SUBAPPLICATION VDS_Auswahl (* Waehlt per Button die satellitengestuetzte Geschwindigkeit (VDS) als Quelle aus, merkt sich die Auswahl persistent im NVS, setzt bei Auswahl die anderen Quellen zurueck und liefert die VDS-Sensordaten nach aussen *)
  (* Standard: 61499-2 *)
  (* Version 1.0, 2026-08-27, Franz *)
  PACKAGE FBs::Baumsetzer::func::Automatik;
  IMPORT NVS_Keys::Key_VDS_Store;
  IMPORT isobus::UT::io::Button::ButtonActivationCode::BT_RELEASED_UNLATCHED;
  IMPORT test::FBs::Baumsetzer::Constants::DefaultPool::Button_VDS;
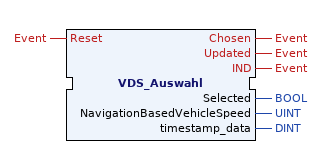
  EVENT_INPUT
    Reset; (* Anforderung von einer der anderen Quellen: eigene Auswahl zuruecksetzen *)
  END_EVENT
  EVENT_OUTPUT
    Chosen; (* Button_VDS wurde gedrueckt: eigene Auswahl setzen und alle anderen Quellen zuruecksetzen *)
    Updated; (* Ausgewaehlt-Status verfuegbar bzw. geaendert (Init-Lesen oder Aenderung); Trigger fuer nachgelagerte Verarbeitung (u.a. Hintergrundfarbe) *)
    IND; (* Neue VDS-Daten empfangen (Indication von I_VDS) *)
  END_EVENT
  VAR_OUTPUT
    Selected : BOOL; (* TRUE wenn VDS aktuell als Geschwindigkeitsquelle ausgewaehlt ist *)
    NavigationBasedVehicleSpeed : UINT; (* Satellitengestuetzte Fahrzeuggeschwindigkeit (PGN 65256, SPN 517) *)
    timestamp_data : DINT; (* Zeitstempel der letzten VDS-Botschaft *)
  END_VAR
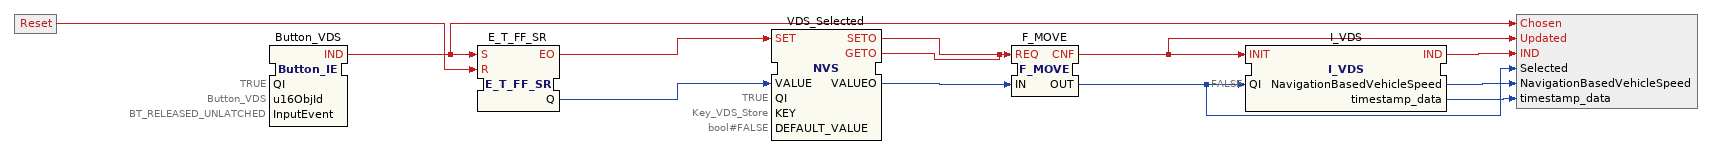
  FBS
    Button_VDS : isobus::UT::io::Button::Button_IE(QI := TRUE, u16ObjId := Button_VDS, InputEvent := BT_RELEASED_UNLATCHED);
    E_T_FF_SR : iec61499::events::E_T_FF_SR;
    VDS_Selected : logiBUS::storage::esp32_nvs::NVS(QI := TRUE, KEY := Key_VDS_Store, DEFAULT_VALUE := bool#FALSE);
    F_MOVE : iec61131::selection::F_MOVE; {SET_ATTRIBUTE(DataType, BOOL)}
    I_VDS : isobus::tecu::I_VDS(QI := FALSE);
  END_FBS
  EVENT_CONNECTIONS
    Button_VDS.IND TO E_T_FF_SR.S;
    Button_VDS.IND TO Chosen;
    Reset TO E_T_FF_SR.R;
    E_T_FF_SR.EO TO VDS_Selected.SET;
    VDS_Selected.SETO TO F_MOVE.REQ;
    VDS_Selected.GETO TO F_MOVE.REQ;
    F_MOVE.CNF TO I_VDS.INIT;
    F_MOVE.CNF TO Updated;
    I_VDS.IND TO IND;
  END_CONNECTIONS
  DATA_CONNECTIONS
    E_T_FF_SR.Q TO VDS_Selected.VALUE;
    VDS_Selected.VALUEO TO F_MOVE.IN;
    F_MOVE.OUT TO I_VDS.QI;
    F_MOVE.OUT TO Selected;
    I_VDS.NavigationBasedVehicleSpeed TO NavigationBasedVehicleSpeed;
    I_VDS.timestamp_data TO timestamp_data;
  END_CONNECTIONS
END_SUBAPPLICATION
